Staubli VAL3: SE.pgx

public program SE(dio x_dInput, dio x_dOutput, num x_nLength)
begin

  //"set delay"
  //set the x_dOutput only when x_dInput is true for a time greater than x_nLength
  //note: x_dInput isn't necessarily an input

  if taskStatus("SE_"+toString("",nSE_Count))==-1
    taskCreate "SE_"+toString("",nSE_Count),10,exeSE(x_dInput,x_dOutput,x_nLength)
    nSE_Count=nSE_Count+1
    if nSE_Count>nMaxTask
      nSE_Count=0
    endIf
  else
    logMsg("libSignals/SE->can't create SE task")
  endIf

end
